{attribute 'GeneratedUsingTerminal: EP9521-0020-0000'}
{attribute addProperty BoxType "EP9521-0020-0000"}
{attribute addProperty Description "EP9521-0020 MediaConverter for EtherCAT Box Modules (FX-MultiMode)"}
{attribute addProperty Physics "YYY"}
{attribute addProperty Id "InfoDataAT %I*InfoData_6F19DB2B2"}
{attribute addProperty CRC "532711307"}
{attribute addProperty Size "2"}
TYPE EP9521_1FC0878B EXTENDS EtcSlaveBoxBase_77A0E4A7 :
STRUCT
	{attribute addProperty Name "InfoData"}
	InfoData : InfoData_6F19DB2B;
END_STRUCT
END_TYPE

(* stored: Version 1.2.0.0, ProductVersion 3.1.4024.9
   DUT EP9521_1FC0878B: Id {f6c5dd3a-b5d6-4c09-9798-edb52660740c} *)
